{attribute 'linkalways'} 
{attribute 'no_explicit_call' := 'This FB is a CLASS and must be accessed using methods or properties'}
{attribute 'enable_dynamic_creation'}
FUNCTION_BLOCK Node_F_VN_ContourExtremePoint EXTENDS VisionNode
VAR
    ipContour : _ITcVnContainer;
    eDirection : _ETcVnExtremePointDirection(ETcVnExtremePointDirection.TCVN_EPD_TOP_LEFT);
    aExtremePoint : _TcVnPoint2_LREAL;
    hrPrev : _HRESULT(S_OK);
	hresult : _HRESULT(S_OK);
END_VAR

METHOD PUBLIC  Clone : I_Node
VAR
	pNode : POINTER TO Node_F_VN_ContourExtremePoint;
END_VAR
pNode := __NEW(Node_F_VN_ContourExtremePoint);
Clone := pNode^;
END_METHOD

METHOD FB_init : BOOL
VAR_INPUT
	bInitRetains : BOOL; // if TRUE, the retain variables are initialized (warm start / cold start)
	bInCopyCode : BOOL;  // if TRUE, the instance afterwards gets moved into the copy code (online change)
END_VAR
AddInput('ipContour', ipContour);
AddParameter('eDirection', eDirection);
AddInput('hrPrev', hrPrev);
AddOutput('aExtremePoint', aExtremePoint);
AddOutput('hresult',hresult);
END_METHOD

METHOD PROTECTED OnExecute
hresult.Value := F_VN_ContourExtremePoint(
	ipContour := ipContour.Value,
    eDirection := eDirection.Value,
    aExtremePoint := aExtremePoint.Value,
	hrPrev:= hrPrev.Value);
END_METHOD

METHOD PUBLIC PreExecutionCheck
VAR_INPUT
	Check : I_PreExecutionChecks;
END_VAR
Check.IsTrue((ipContour.IsType(TC_GLOBAL_CONST_LIST.ContainerType_Vector_TcVnPoint2_DINT) OR
              ipContour.IsType(TC_GLOBAL_CONST_LIST.ContainerType_Vector_TcVnPoint2_REAL) OR
              ipContour.IsType(TC_GLOBAL_CONST_LIST.ContainerType_Vector_TcVnPoint2_LREAL)),
              'ipContour contains incorrect type');
END_METHOD

END_FUNCTION_BLOCK

(* stored: Version 1.1.0.1, ProductVersion 3.1.4026.13
   POU Node_F_VN_ContourExtremePoint: Id {b4fa4d6c-571d-08f4-12c2-9a865ffb2c0d}, SpecialFunc None
   Folder Constructor: Id {8e777ee0-8702-0a88-3994-fe309b02e4f8}
   Method Clone: Id {7a174f11-f55b-0c2a-2b06-ffdf7f9d6c0e}
   Method FB_init: Id {7aa3ebe6-812a-0974-0f09-6555c1ffc788}
   Method OnExecute: Id {068630b0-0fa4-0456-1581-9ef662f57a4d}
   Method PreExecutionCheck: Id {3ae936df-7885-0292-184c-d5880080e7d7} *)
